FUNCTION_BLOCK L3_CompletedSetupHDLR (* Basic Function Block Type *)
  (* Standard: 61499-2 *)
  (* Version 0.0, 2014-11-03, EQUEROL, UJI *)
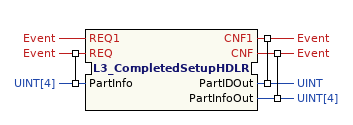
  EVENT_INPUT
    REQ1; (* Completed parts request *)
    REQ WITH PartInfo; (* Normal execution request *)
  END_EVENT
  EVENT_OUTPUT
    CNF1 WITH PartIDOut; (* Conpleted setup request confirmation *)
    CNF WITH PartInfoOut; (* Execution confirmation *)
  END_EVENT
  VAR_INPUT
    PartInfo : ARRAY [0..3] OF UINT; (* Part identifier, Family and type *)
  END_VAR
  VAR_OUTPUT
    PartIDOut : UINT; (* Part identifier *)
    PartInfoOut : ARRAY [0..3] OF UINT;
  END_VAR
  VAR
    PartBuffer : ARRAY [0..14] OF UINT := [0,0,0,0,0,0,0,0,0,0,0,0,0,0,0]; (* Buffer to hold received "parts" i.e parts which setups have been completed; FIFO discipline *)
    TailIndex : USINT := 0; (* Position within the buffer where next part to be send is stock *)
    HeadIndex : USINT := 0; (* Poisiton within the buffer where next completed part will be stock *)
    BufferSize : USINT := 15; (* const buffer size *)
  END_VAR
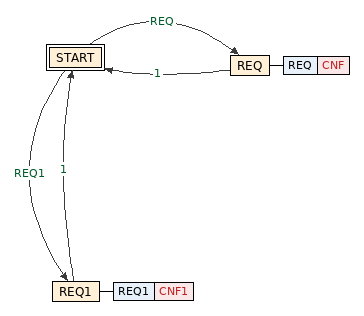
  EC_STATES
    START; (* Initial State *)
    REQ : REQ -> CNF; (* Normal execution *)
    REQ1 : REQ1 -> CNF1;
  END_STATES
  EC_TRANSITIONS
    START TO REQ := REQ;
    START TO REQ1 := REQ1;
    REQ TO START := 1;
    REQ1 TO START := 1;
  END_TRANSITIONS
  ALGORITHM REQ IN ST: (* Normally executed algorithm *)
(*Stack the received part*)
PartBuffer[HeadIndex] := PartInfo[0];

(*PostIncrement HeadIndex*)
HeadIndex := HeadIndex + 1;
IF HeadIndex >= BufferSize THEN
	(*HeadIndex =% 15*)
	HeadIndex := 0;
END_IF;

(*Check if buffer is full*)
IF HeadIndex = TailIndex THEN
	(*Buffer is full, HeadIndex can't be incremented*)
	IF HeadIndex = 0 THEN
		HeadIndex := BufferSize -1;
	ELSE
		HeadIndex := HeadIndex - 1;
	END_IF;
END_IF;

(*Map the response to the right machine*)
PartInfoOut[0] := PartInfo[0];
PartInfoOut[1] := PartInfo[1];
PartInfoOut[2] := PartInfo[2];
PartInfoOut[3] := PartInfo[3];
  END_ALGORITHM
  ALGORITHM REQ1 IN ST: (* Completed part request *)
IF HeadIndex = TailIndex THEN
	(*Buffer is empty*)
	PartIDOut := 0;
ELSE
	PartIDOut := PartBuffer[TailIndex];
	(*Increase tail index*)
	TailIndex := TailIndex + 1;
	IF TailIndex >= BufferSize THEN
		(* TaiIndex =% 15*)
		TailIndex := 0;
	END_IF;
END_IF;
  END_ALGORITHM
END_FUNCTION_BLOCK
